TYPE ST_MagnetControl :
STRUCT
END_STRUCT
END_TYPE

(* stored: Version 1.1.0.1, ProductVersion 3.1.4024.12
   DUT ST_MagnetControl: Id {e2e1ef87-de1e-4e6a-a268-1fa4c2299d10} *)
